// Mitsubishi GX Works2 project: FX2   PLC: FX2/FX2C

PROGRAM MAIN
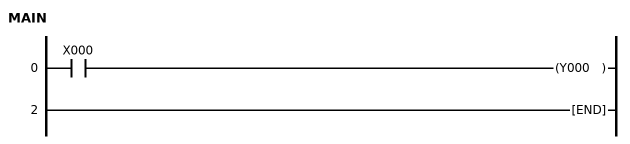
0     LD      X000
      OUT     Y000
2     END
END_PROGRAM
